Staubli VAL3: getItem.pgx

public program getItem(string& x_sItem, string& x_sId)
begin
  // get the name
  x_sItem=saveInOut:dOutput[x_sId].sName
end
